# B&R Automation Studio project Task2
Automation Studio 4.9

## Logical view

### Global.typ - Global data types
```iecst
TYPE
	Sys_Handler : 	STRUCT
		Initialize:BOOL:=FALSE;
		Run:BOOL:=FALSE;
		On_Phase_Stop:BOOL:=FALSE;
	END_STRUCT;

	Sub_Sys_Handler : 	STRUCT
		Initialize:BOOL:=FALSE;
		Enable:BOOL:=FALSE;
		Disable:BOOL:=FALSE;
		On_Phase_Stop:BOOL:=FALSE;
	END_STRUCT;

END_TYPE
```

### Global.var - Global variables
```iecst
(* Generic-Axis *)
VAR
	gConveyor : ACP10AXIS_typ;
	gKnife : ACP10AXIS_typ;
END_VAR

(* Logical Buttons*)
VAR
	Init_logical : BOOL;
	Start_logical : BOOL;
	On_Phase_Stop_logical : BOOL;
	Trigger_logical : BOOL;
	Reset_logical : BOOL;
END_VAR
(* Handlers *)
VAR
	Machine_Handler : Sys_Handler;
	Conveyor_Handler : Sub_Sys_Handler;
	Cutter_Handler : Sub_Sys_Handler;
	Signal_Management_Handler : Sys_Handler;
END_VAR

VAR
	CONVEYOR_VELOCITY : REAL := 100;
	CONVEYOR_MAX_VELOCITY : REAL := 100;
	CUTTER_VELOCITY : REAL := 400;
	CUTTER_MAX_VELOCITY : REAL := 400;
END_VAR
```

### Package Logical/Libraries - Global libraries

### Library Logical/Libraries/gAxis_lib (IEC)

#### Types.typ - Exported data types
```iecst
TYPE
	gAxis_StateType :
		(
		NotPowered,
		WaitPower,
		Powered,
		Ready,
		CommandHandler,
		MoveVelocity,
		CheckVelocity,
		MoveAdditive,
		CheckPosition,
		CamInState,
		CheckCamState,
		Stop
		);
END_TYPE
```

#### Constants.var - Exported constants
```iecst
VAR CONSTANT
	AXIS_NULL_COMMAND : WORD := 0;
	AXIS_MOVE_VELOCITY : WORD := 1;
	AXIS_MOVE_ADDITIVE : WORD := 2;
	AXIS_CAM_IN : WORD := 3;
	AXIS_STOP : WORD := 4;
	STANDSTILL : WORD := 5;
	DISCRETE_MOTION : WORD := 6;
	CONTINOUS_MOTION : WORD := 7;
END_VAR
```

#### gAxis_lib.fun - Exported functions and function blocks
```iecst
FUNCTION_BLOCK gAxis (*TODO: Add your comment here*) (*$GROUP=User,$CAT=User,$GROUPICON=User.png,$CATICON=User.png*)
	VAR_INPUT
		Master : UDINT;
		Slave : UDINT;
		AxisOperation : INT;
		AxisCommand : WORD := 777;
		Distance : REAL;
		Position : REAL;
		Velocity : REAL;
		Acceleration : REAL;
		Deceleration : REAL;
		Jerk : REAL;
		Direction : USINT;
		ArraySize : INT;
		Scale : REAL;
		Offset : REAL;
		RatioNumerator : INT;
		RatioDenominator : INT;
		CamTableID : USINT;
		MasterScaling : REAL := 360;
		SlaveScaling : REAL := 360;
		MasterOffset : REAL := 10;
		SlaveOffset : REAL := 0;
		StartMode : USINT := 1; (*mcRELATIVE*)
		AxisEnable_in : BOOL;
		Reset : BOOL;
	END_VAR
	VAR_OUTPUT
		ActualPosition : REAL;
		ActualVelocity : REAL;
		AxisEnable_out : BOOL;
		CommandExecuted : BOOL := FALSE;
		CommandAborted : BOOL;
		AxisStatus : WORD;
		AxisError : BOOL;
		AxisErrorID : WORD;
		AxisNotInizialized : BOOL;
	END_VAR
	VAR
		INIT : INT;
		RUN : INT;
		OldDistance : REAL;
		OldVelocity : REAL;
		OldCamTableID : USINT;
		AxisState : gAxis_StateType := NotPowered;
		gA_Power : MC_Power;
		gA_Home : MC_Home;
		gA_MoveVelocity : MC_MoveVelocity;
		gA_MoveAdditive : MC_MoveAdditive;
		gA_CamIn : MC_CamIn;
		gA_CamOut : MC_CamOut;
		gA_ReadActualPosition : MC_ReadActualPosition;
		gA_ReadActualVelocity : MC_ReadActualVelocity;
		gA_ReadAxisError : MC_ReadAxisError;
		gA_ReadStatus : MC_ReadStatus;
		gA_Stop : MC_Stop;
	END_VAR
END_FUNCTION_BLOCK
```

#### gAxis.st
```iecst
(* TODO: Add your comment here *)
FUNCTION_BLOCK gAxis

	CASE AxisState OF

		NotPowered:
			IF AxisEnable_in THEN
				gA_Power.Enable := TRUE;
				AxisState := WaitPower;
			END_IF;

		WaitPower:
			IF gA_Power.Status THEN
				gA_Home.Execute := TRUE;
				(*gA_CamTableSelect.Execute := TRUE;*)
				AxisState := Powered;
			END_IF

		Powered:
			(*IF gA_Home.Done AND gA_CamTableSelect.Done THEN*)

			IF gA_Home.Done THEN
				gA_Home.Execute := FALSE;
				AxisEnable_out := FALSE;
				AxisState := Ready;
			END_IF;

		Ready:
			IF AxisCommand = AXIS_MOVE_VELOCITY THEN
				CommandExecuted := FALSE;
				gA_MoveVelocity.Velocity := Velocity;
				gA_MoveVelocity.Execute := TRUE;
				AxisState := MoveVelocity;
			END_IF;

			IF AxisCommand = AXIS_MOVE_ADDITIVE THEN
				CommandExecuted := FALSE;
				gA_MoveAdditive.Distance := Distance;
				gA_MoveAdditive.Execute := TRUE;
				AxisState := MoveAdditive;
			END_IF;

			IF AxisCommand = AXIS_CAM_IN THEN
				CommandExecuted := FALSE;
				gA_CamIn.Execute := TRUE;
				AxisState := CamInState;
			END_IF

			IF AxisCommand = AXIS_STOP THEN
				CommandExecuted := FALSE;
				gA_Stop.Execute := TRUE;
				AxisState := Stop;
			END_IF;

		MoveVelocity:
			IF gA_MoveVelocity.InVelocity THEN
				OldVelocity := Velocity;
				gA_MoveVelocity.Execute := FALSE;
				CommandExecuted := TRUE;
				AxisState := CheckVelocity;
			END_IF;

			IF AxisCommand <> AXIS_MOVE_VELOCITY THEN
				gA_MoveVelocity.Execute := FALSE;
				CommandExecuted := FALSE;
				AxisState := Ready;
			END_IF;

		CheckVelocity:
			IF Velocity <> OldVelocity THEN
				OldVelocity := Velocity;
				gA_MoveVelocity.Velocity := Velocity;
				gA_MoveVelocity.Execute := TRUE;
				CommandExecuted := FALSE;
				AxisState := MoveVelocity;
			END_IF;

			IF AxisCommand <> AXIS_MOVE_VELOCITY THEN
				gA_MoveVelocity.Execute := FALSE;
				CommandExecuted := FALSE;
				AxisState := Ready;
			END_IF;

		MoveAdditive:
			IF gA_MoveAdditive.Done THEN
				OldDistance := Distance;
				gA_MoveAdditive.Execute := FALSE;
				CommandExecuted := TRUE;
				AxisState := CheckPosition;
			END_IF;

			IF AxisCommand <> AXIS_MOVE_ADDITIVE THEN
				gA_MoveAdditive.Execute := FALSE;
				CommandExecuted := FALSE;
				AxisState := Ready;
			END_IF;

		CheckPosition:
			IF Distance <> OldDistance THEN
				OldDistance := Distance;
				gA_MoveAdditive.Distance := Distance;
				gA_MoveAdditive.Execute := TRUE;
				CommandExecuted := FALSE;
				AxisState := MoveAdditive;
			END_IF;

			IF AxisCommand <> AXIS_MOVE_ADDITIVE THEN
				gA_MoveAdditive.Execute := FALSE;
				CommandExecuted := FALSE;
				AxisState := Ready;
			END_IF;

		CamInState:
			IF gA_CamIn.EndOfProfile THEN
				OldCamTableID := CamTableID;
				gA_CamIn.Execute := FALSE;
				CommandExecuted := TRUE;
				AxisState := CheckCamState;
			END_IF

			IF AxisCommand <> AXIS_CAM_IN THEN
				gA_CamIn.Execute := FALSE;
				CommandExecuted := FALSE;
				AxisState :=  Ready;
			END_IF

		CheckCamState:
			IF CamTableID <> OldCamTableID THEN
				OldCamTableID := CamTableID;
				gA_CamIn.Execute := TRUE;
				CommandExecuted := FALSE;
				AxisState := CamInState;
			END_IF;

			IF AxisCommand <> AXIS_MOVE_ADDITIVE THEN
				gA_CamIn.Execute := FALSE;
				CommandExecuted := FALSE;
				AxisState := Ready;
			END_IF;

		Stop:
			IF (gA_Stop.Done) THEN
				CommandExecuted := TRUE;
			END_IF

			IF (AxisCommand <> AXIS_STOP ) THEN
				gA_Stop.Execute := FALSE;
				CommandExecuted := FALSE;

				AxisState := Ready;
			END_IF

	END_CASE;

	AxisEnable_in := AxisEnable_out;

	gA_Power.Axis := Slave;
	gA_Power();

	gA_Home.Axis := Slave;
	gA_Home.Position := Position;
	gA_Home();

	(*
	gA_CamTableSelect.Master := Master;
	gA_CamTableSelect.Slave := Slave;
	gA_CamTableSelect.CamTable := 'Cam';
	gA_CamTableSelect.Periodic := mcNON_PERIODIC;
	gA_CamTableSelect();
	CamTableID := gA_CamTableSelect.CamTableID;
	*)

	gA_MoveVelocity.Axis := Slave;
	gA_MoveVelocity.Velocity := Velocity;
	gA_MoveVelocity.Acceleration := Acceleration;
	gA_MoveVelocity.Deceleration := Deceleration;
	gA_MoveVelocity();

	IF OldDistance = 0 THEN
		OldDistance := Distance;
	END_IF;

	gA_MoveAdditive.Axis := Slave;
	gA_MoveAdditive.Distance := Distance;
	gA_MoveAdditive.Velocity := Velocity;
	gA_MoveAdditive.Acceleration := Acceleration;
	gA_MoveAdditive.Deceleration := Deceleration;
	gA_MoveAdditive();

	gA_ReadActualPosition.Axis := Slave;
	gA_ReadActualPosition.Enable := TRUE;
	gA_ReadActualPosition();

	ActualPosition := gA_ReadActualPosition.Position;

	gA_ReadActualVelocity.Axis := Slave;
	gA_ReadActualVelocity.Enable := TRUE;
	gA_ReadActualVelocity();

	ActualVelocity := gA_ReadActualVelocity.Velocity;

	gA_CamIn.CamTableID := CamTableID;
	gA_CamIn.StartMode := StartMode;
	gA_CamIn.MasterScaling := MasterScaling;
	gA_CamIn.SlaveScaling := SlaveScaling;
	gA_CamIn.MasterOffset := MasterOffset;
	gA_CamIn.SlaveOffset := SlaveOffset;
	gA_CamIn(Master := Master, Slave := Slave);

	gA_CamOut(Slave:=Slave);

	gA_Stop.Axis := Slave;
	gA_Stop.Deceleration := Deceleration;
	gA_Stop();

	gA_ReadStatus.Enable := TRUE;
	gA_ReadStatus.Axis := Slave;
	gA_ReadStatus();

	IF gA_ReadStatus.StandStill THEN
		AxisStatus := STANDSTILL;
	END_IF;

	IF gA_ReadStatus.DiscreteMotion THEN
		AxisStatus := DISCRETE_MOTION;
	END_IF;

	IF gA_ReadStatus.ContinuousMotion THEN
		AxisStatus := CONTINOUS_MOTION;
	END_IF;

END_FUNCTION_BLOCK
```

### Library Logical/Libraries/filter_lib (IEC)

#### filter.st
```iecst
(* TODO: Add your comment here *)
FUNCTION_BLOCK filter

	IF Delay > 0 THEN
		Delay := Delay -1;
	END_IF;

	IF Delay = 0 THEN
	  DelayedSignal := Signal;
	END_IF;

	IF Signal = DelayedSignal THEN

		IF Signal THEN
			Delay := DeactivationDelay;
		ELSE
			Delay := ActivationDelay;
		END_IF;

	END_IF;
END_FUNCTION_BLOCK
```

- Visualisation Logical/mappView (not shown)


- Data object Logical/gConveyorobj/gConveyora (Apt) (no source held here)

### Package Logical/gKnifeobj - gKnifeobj

- Data object Logical/gKnifeobj/gKnifea (Apt) (no source held here)

### Data object Logical/gKnifeobj/gKnifei (Ax)

#### gKnifei.ax
```
InitParameter (Version=5.16.2, NcSwId=Acp10)
  ACP10AXIS_typ:
    dig_in:
      level:
        reference = ncACTIV_HI
        pos_hw_end = ncACTIV_HI
        neg_hw_end = ncACTIV_HI
        trigger1 = ncACTIV_HI
        trigger2 = ncACTIV_HI
    encoder_if:
      parameter:
        count_dir = ncSTANDARD
        scaling:
          load:
            units = 360
            rev_motor = 1
    limit:
      parameter:
        v_pos = 10000
        v_neg = 10000
        a1_pos = 50000
        a2_pos = 50000
        a1_neg = 50000
        a2_neg = 50000
        t_jolt = 0
        t_in_pos = 0
        pos_sw_end = 2000000000
        neg_sw_end = -2000000000
        ds_warning = 500
        ds_stop = 1000
        a_stop = 1.0e30
        dv_stop = 0
        dv_stop_mode = ncOFF
    controller:
      mode = ncPOSITION
      position:
        kv = 50
        tn = 0
        t_predict = 0.0004
        t_total = 0.0004
        p_max = 1.0e30
        i_max = 0
      speed:
        kv = 2.0
        tn = 0
        t_filter = 0.0
        isq_filter1:
          type = ncOFF
          a0 = 0.0
          a1 = 0.0
          b0 = 0.0
          b1 = 0.0
          b2 = 0.0
          c0_par_id = 0
          c1_par_id = 0
        isq_filter2:
          type = ncOFF
          a0 = 0.0
          a1 = 0.0
          b0 = 0.0
          b1 = 0.0
          b2 = 0.0
          c0_par_id = 0
          c1_par_id = 0
        isq_filter3:
          type = ncOFF
          a0 = 0.0
          a1 = 0.0
          b0 = 0.0
          b1 = 0.0
          b2 = 0.0
          c0_par_id = 0
          c1_par_id = 0
      uf:
        type = ncLINEAR + ncCORRECTION
        auto_config = ncMOTOR_PAR
        u0 = 0
        un = 0
        fn = 50.0
        k_f_slip = 0
      ff:
        mode = ncSTANDARD
        torque_load = 0.0
        torque_pos = 0.0
        torque_neg = 0.0
        kv_torque = 0.0
        inertia = 0.0
        t_filter_a = 0.0
      fb:
        mode = ncSTANDARD
        speed_mix_ratio = 0.0
        speed_kv = 2.0
      model:
        mass1:
          inertia = 0
          viscous_friction = 0
        mass2:
          inertia = 0
          viscous_friction = 0
          stiffness = 0
          damping = 0
    move:
      stop:
        parameter[0]:
          decel_ramp = ncA_LIMIT
          controller = ncON
        parameter[1]:
          decel_ramp = ncA_LIMIT
          controller = ncON
        parameter[2]:
          decel_ramp = ncA_LIMIT
          controller = ncON
        parameter[3]:
          decel_ramp = ncA_LIMIT
          controller = ncON
        quickstop:
          decel_ramp = ncA_LIMIT
          t_jolt = 0
        drive_error:
          decel_ramp = ncA_LIMIT
      homing:
        parameter:
          s = 0
          v_switch = 5000
          v_trigger = 500
          a = 50000
          mode = ncDIRECT
          edge_sw = ncPOSITIVE
          start_dir = ncPOSITIVE
          trigg_dir = ncPOSITIVE
          ref_pulse = ncOFF
          fix_dir = ncOFF
          tr_s_block = 0
          torque_lim = 0
          ds_block = 0
          ds_stop = 0
      basis:
        parameter:
          v_pos = 5000
          v_neg = 5000
          a1_pos = 50000
          a2_pos = 50000
          a1_neg = 50000
          a2_neg = 50000
    message:
      text:
        parameter:
          format = ncBREAK
          columns = 80
          data_modul = acp10etxen
```

### Data object Logical/Cam (Cam)

#### Cam.cam
```
CamProfile (NcSwId=ACP10, MasterAxisVelocity=1, MasterAxisAcceleration=0, DefaultCurveType=Polynomial5, MathematicalNotation=true)
  FixPoint (x=0, IsMathX=true, y=0, IsDefinedDy=false, Dy=0, IsMathDy=true, IsDefinedDdy=false, Ddy=0, IsMathDdy=true, IsDefinedDddy=false, Dddy=0, IsMathDddy=true)
  FixPoint (x=0.5, IsMathX=true, y=0, IsDefinedDy=false, Dy=0, IsMathDy=true, IsDefinedDdy=false, Ddy=0, IsMathDdy=true, IsDefinedDddy=false, Dddy=0, IsMathDddy=true)
  FixPoint (x=0.55, IsMathX=true, y=0.5, IsDefinedDy=false, Dy=0, IsMathDy=true, IsDefinedDdy=false, Ddy=0, IsMathDdy=true, IsDefinedDddy=false, Dddy=0, IsMathDddy=true)
  FixPoint (x=0.6, IsMathX=true, y=0, IsDefinedDy=false, Dy=0, IsMathDy=true, IsDefinedDdy=false, Ddy=0, IsMathDdy=true, IsDefinedDddy=false, Dddy=0, IsMathDddy=true)
  FixPoint (x=1, IsMathX=true, y=0, IsDefinedDy=false, Dy=0, IsMathDy=true, IsDefinedDdy=false, Ddy=0, IsMathDdy=true, IsDefinedDddy=false, Dddy=0, IsMathDddy=true)
  Curve (Type=Polynomial5)
    LeftBoundary (IsDefinedDdy=false, Ddy=0, IsMathDdy=true, IsDefinedDddy=false, Dddy=0, IsMathDddy=true)
    RightBoundary (IsDefinedDdy=false, Ddy=0, IsMathDdy=true, IsDefinedDddy=false, Dddy=0, IsMathDddy=true)
    Spline3 (IsContinuous4Derivative=false, IsDefinedSaddlePoint=false, IsDefinedLineAs2ndSegment=false, IsDefinedSlopeOfLine=false, SlopeOfLine=0, IsMathSlopeOfLine=true)
    Supremum (y=1.7e+308, Dy=1.7e+308, IsMathDy=true, Ddy=1.7e+308, IsMathDdy=true, Dddy=1.7e+308, IsMathDddy=true)
    Infimum (y=-1.7e+308, Dy=-1.7e+308, IsMathDy=true, Ddy=-1.7e+308, IsMathDdy=true, Dddy=-1.7e+308, IsMathDddy=true)
  Curve (Type=Polynomial5)
    LeftBoundary (IsDefinedDdy=false, Ddy=0, IsMathDdy=true, IsDefinedDddy=false, Dddy=0, IsMathDddy=true)
    RightBoundary (IsDefinedDdy=false, Ddy=0, IsMathDdy=true, IsDefinedDddy=false, Dddy=0, IsMathDddy=true)
    Spline3 (IsContinuous4Derivative=false, IsDefinedSaddlePoint=false, IsDefinedLineAs2ndSegment=false, IsDefinedSlopeOfLine=false, SlopeOfLine=0, IsMathSlopeOfLine=true)
    Supremum (y=1.7e+308, Dy=1.7e+308, IsMathDy=true, Ddy=1.7e+308, IsMathDdy=true, Dddy=1.7e+308, IsMathDddy=true)
    Infimum (y=-1.7e+308, Dy=-1.7e+308, IsMathDy=true, Ddy=-1.7e+308, IsMathDdy=true, Dddy=-1.7e+308, IsMathDddy=true)
  Curve (Type=Polynomial5)
    LeftBoundary (IsDefinedDdy=false, Ddy=0, IsMathDdy=true, IsDefinedDddy=false, Dddy=0, IsMathDddy=true)
    RightBoundary (IsDefinedDdy=false, Ddy=0, IsMathDdy=true, IsDefinedDddy=false, Dddy=0, IsMathDddy=true)
    Spline3 (IsContinuous4Derivative=false, IsDefinedSaddlePoint=false, IsDefinedLineAs2ndSegment=false, IsDefinedSlopeOfLine=false, SlopeOfLine=0, IsMathSlopeOfLine=true)
    Supremum (y=1.7e+308, Dy=1.7e+308, IsMathDy=true, Ddy=1.7e+308, IsMathDdy=true, Dddy=1.7e+308, IsMathDddy=true)
    Infimum (y=-1.7e+308, Dy=-1.7e+308, IsMathDy=true, Ddy=-1.7e+308, IsMathDdy=true, Dddy=-1.7e+308, IsMathDddy=true)
  Curve (Type=Polynomial5)
    LeftBoundary (IsDefinedDdy=false, Ddy=0, IsMathDdy=true, IsDefinedDddy=false, Dddy=0, IsMathDddy=true)
    RightBoundary (IsDefinedDdy=false, Ddy=0, IsMathDdy=true, IsDefinedDddy=false, Dddy=0, IsMathDddy=true)
    Spline3 (IsContinuous4Derivative=false, IsDefinedSaddlePoint=false, IsDefinedLineAs2ndSegment=false, IsDefinedSlopeOfLine=false, SlopeOfLine=0, IsMathSlopeOfLine=true)
    Supremum (y=1.7e+308, Dy=1.7e+308, IsMathDy=true, Ddy=1.7e+308, IsMathDdy=true, Dddy=1.7e+308, IsMathDddy=true)
    Infimum (y=-1.7e+308, Dy=-1.7e+308, IsMathDy=true, Ddy=-1.7e+308, IsMathDdy=true, Dddy=-1.7e+308, IsMathDddy=true)
  Cam (LeftBoundaryIndex=0, RightBoundaryIndex=4)
    Supremum (y=1.7e+308, Dy=1.7e+308, IsMathDy=true, Ddy=1.7e+308, IsMathDdy=true, Dddy=1.7e+308, IsMathDddy=true)
    Infimum (y=-1.7e+308, Dy=-1.7e+308, IsMathDy=true, Ddy=-1.7e+308, IsMathDdy=true, Dddy=1.7e+308, IsMathDddy=true)
  ChartExtensions
```

### Program Logical/Main (IEC)

#### Types.typ
```iecst
TYPE
	Main_States: (
		Main_ready_to_be_initialized,
		Main_initializing,
		Main_ready_to_run,
		Main_running,
		Main_on_phase_stopping
	);
END_TYPE
```

#### Main.st
```iecst
PROGRAM _CYCLIC
	(* Insert code here *)

	CASE state OF
		Main_ready_to_be_initialized:
			IF Init_logical THEN
				Machine_Handler.Initialize := TRUE;

				state := Main_initializing;
			END_IF;

		Main_initializing:
			IF NOT Machine_Handler.Initialize THEN

				state := Main_ready_to_run;
			END_IF;

		Main_ready_to_run:
			IF Start_logical THEN
				Machine_Handler.Run := TRUE;

				state := Main_running;
			END_IF;

		Main_running:
			IF On_Phase_Stop_logical THEN
				Machine_Handler.Run := FALSE;
				Machine_Handler.On_Phase_Stop := TRUE;

				state := Main_on_phase_stopping;
			END_IF;

		Main_on_phase_stopping:
			IF NOT On_Phase_Stop_logical THEN
				Machine_Handler.On_Phase_Stop := FALSE;

				state := Main_ready_to_run;
			END_IF;
	END_CASE;

END_PROGRAM
```

### Program Logical/MachineProgram (IEC)

#### Types.typ
```iecst
TYPE
	Machine_States: (
					Machine_ready_to_be_initialized,
					Machine_initializing,
					Machine_ready_to_run,
					Conveyor_Enabling,
					Cutter_Enabling,
					Machine_on_phase_stopping);
END_TYPE
```

#### Variables.var
```iecst
VAR
	state: Machine_States := Machine_ready_to_be_initialized;
END_VAR
```

#### Main.st
```iecst
PROGRAM _CYCLIC
	(* Insert code here *)
	CASE state OF

		Machine_ready_to_be_initialized:
			IF Machine_Handler.Initialize THEN
				Conveyor_Handler.Initialize := TRUE;
				Cutter_Handler.Initialize := TRUE;

				state := Machine_initializing;
			END_IF;

		Machine_initializing:
			IF NOT Conveyor_Handler.Initialize AND NOT Cutter_Handler.Initialize THEN
				Machine_Handler.Initialize := FALSE;

				state := Machine_ready_to_run;
			END_IF;

		Machine_ready_to_run:
			IF Machine_Handler.Run THEN
				Conveyor_Handler.Enable := TRUE;

				state := Conveyor_Enabling;
			END_IF;

		Conveyor_Enabling:
			IF Machine_Handler.On_Phase_Stop THEN
				Conveyor_Handler.On_Phase_Stop := TRUE;
				Cutter_Handler.On_Phase_Stop := TRUE;

				state := Machine_on_phase_stopping;

			ELSIF NOT Conveyor_Handler.Enable AND Trigger_logical THEN
				Cutter_Handler.Enable := TRUE;

				state := Cutter_Enabling;
			END_IF;

		Cutter_Enabling:
			IF NOT Cutter_Handler.Enable THEN

				state := Conveyor_Enabling;
			END_IF;

		Machine_on_phase_stopping:
			IF NOT Machine_Handler.On_Phase_Stop THEN
				Conveyor_Handler.On_Phase_Stop := FALSE;
				Cutter_Handler.On_Phase_Stop := FALSE;

				state := Machine_ready_to_run;
			END_IF;
	END_CASE;

END_PROGRAM

PROGRAM _EXIT
	(* Insert code here *)

END_PROGRAM
```

### Program Logical/Conveyor (IEC)

#### Types.typ
```iecst
TYPE
	Conveyor_States: (
		Conveyor_ready_to_be_initialized,
		Conveyor_initializing,
		Conveyor_ready_to_be_enabled,
		Conveyor_enabling,
		Conveyor_ready_to_be_disabled,
		Conveyor_on_phase_stopping
	);
END_TYPE
```

#### Variables.var
```iecst
VAR
	Conveyor : gAxis;
END_VAR

VAR
	state: Conveyor_States := Conveyor_ready_to_be_initialized;
END_VAR

VAR
	Axis_Command : WORD := AXIS_NULL_COMMAND;
	Axis_Command_Executed : BOOL;
	Axis_Enable : BOOL;
END_VAR

VAR
	CONVEYOR_POSITION : REAL;
	CONVEYOR_ACTUAL_VELOCITY : INT;
	CONVEYOR_ACCELLERATION : REAL := 100;
	CONVEYOR_DEACCELLERATION : REAL := 100;
	CONVEYOR_DISTANCE : REAL := 100;
END_VAR

VAR CONSTANT
	AXIS_NULL_COMMAND : WORD := 0;
	AXIS_MOVE_VELOCITY : WORD := 1;
	AXIS_MOVE_ADDITIVE : WORD := 2;
	AXIS_CAM_IN : WORD := 3;
	AXIS_STOP : WORD := 4;
END_VAR
```

#### Main.st
```iecst
PROGRAM _INIT
	(* Insert code here *)

END_PROGRAM

PROGRAM _CYCLIC
	(* Insert code here *)
	CASE state OF
		Conveyor_ready_to_be_initialized:
			IF Conveyor_Handler.Initialize THEN
				Axis_Enable := TRUE;

				state := Conveyor_initializing;
			END_IF;

		Conveyor_initializing:
			IF NOT Axis_Enable THEN
				Conveyor_Handler.Initialize := FALSE;

				state := Conveyor_ready_to_be_enabled;
			END_IF;

		Conveyor_ready_to_be_enabled:
			IF Conveyor_Handler.Enable THEN
				Axis_Command := AXIS_MOVE_VELOCITY;

				state := Conveyor_enabling;
			END_IF;

		Conveyor_enabling:
			IF Axis_Command_Executed THEN
				Conveyor_Handler.Enable := FALSE;

				state := Conveyor_ready_to_be_disabled;
			END_IF;

		Conveyor_ready_to_be_disabled:
			IF Conveyor_Handler.On_Phase_Stop THEN
				Axis_Command := AXIS_STOP;

				state := Conveyor_on_phase_stopping;
			END_IF;

		Conveyor_on_phase_stopping:
			IF NOT Conveyor_Handler.On_Phase_Stop THEN

				state := Conveyor_ready_to_be_enabled;
			END_IF;
	END_CASE;

	Conveyor.Slave	:= ADR(gConveyor);

	Conveyor.AxisEnable_in := Axis_Enable;
	Conveyor.AxisCommand := Axis_Command;

	Conveyor.Velocity	:= CONVEYOR_VELOCITY;
	Conveyor.Acceleration	:= CONVEYOR_ACCELLERATION;
	Conveyor.Deceleration	:= CONVEYOR_DEACCELLERATION;

	Conveyor();

	Axis_Enable := Conveyor.AxisEnable_out;
	Axis_Command_Executed := Conveyor.CommandExecuted;
	CONVEYOR_POSITION := Conveyor.ActualPosition;
	CONVEYOR_ACTUAL_VELOCITY := REAL_TO_INT(Conveyor.ActualVelocity);

	ComTCP_SimOutputs.Shaft_0_ACT_POS := CONVEYOR_POSITION;

END_PROGRAM

PROGRAM _EXIT
	(* Insert code here *)

END_PROGRAM
```

### Program Logical/Knife (IEC)

#### Types.typ
```iecst
TYPE
	Cutter_States:
		(
		Cutter_ready_to_be_initialized,
		Cutter_initializing,
		Cutter_ready_to_be_enabled,
		Cutter_enabling
	);
END_TYPE
```

#### Variables.var
```iecst
VAR
	Knife : gAxis;
	CamTableSelect : MC_CamTableSelect;
	CamTableID : USINT;

END_VAR

VAR
	state: Cutter_States := Cutter_ready_to_be_initialized;
END_VAR

VAR
	Axis_Command : WORD := AXIS_NULL_COMMAND;
	Axis_Command_Executed : BOOL;
	Axis_Enable : BOOL;
END_VAR

VAR
	CUTTER_POSITION : REAL;
	CUTTER_ACTUAL_VELOCITY : REAL;
	CUTTER_ACCELLERATION : REAL := 400;
	CUTTER_DEACCELLERATION : REAL := 400;
END_VAR

VAR CONSTANT
	AXIS_NULL_COMMAND : WORD := 0;
	AXIS_MOVE_VELOCITY : WORD := 1;
	AXIS_MOVE_ADDITIVE : WORD := 2;
	AXIS_CAM_IN : WORD := 3;
	AXIS_STOP : WORD := 4;
END_VAR
```

#### Main.st
```iecst
PROGRAM _INIT
	(* Insert code here *)

END_PROGRAM

PROGRAM _CYCLIC
	(* Insert code here *)

	CASE state OF

		Cutter_ready_to_be_initialized:
			IF Cutter_Handler.Initialize THEN
				Axis_Enable := TRUE;
				CamTableSelect.Execute := TRUE;

				state := Cutter_initializing;
			END_IF;

		Cutter_initializing:
			IF NOT Axis_Enable AND CamTableSelect.Done THEN
				Cutter_Handler.Initialize := FALSE;
				CamTableID := CamTableSelect.CamTableID;
				CamTableSelect.Execute := FALSE;

				state := Cutter_ready_to_be_enabled;
			END_IF;

		Cutter_ready_to_be_enabled:
			IF Cutter_Handler.Enable THEN
				Axis_Command := AXIS_CAM_IN;

				state := Cutter_enabling;
			END_IF;

		Cutter_enabling:
			IF Axis_Command_Executed THEN
				Axis_Command := AXIS_NULL_COMMAND;
				Cutter_Handler.Enable := FALSE;

				state := Cutter_ready_to_be_enabled;
			END_IF;

	END_CASE;

	CamTableSelect.Master := ADR(gConveyor);
	CamTableSelect.Slave := ADR(gKnife);
	CamTableSelect.CamTable := 'Cam';
	CamTableSelect.Periodic := mcNON_PERIODIC;
	CamTableSelect();

	Knife.Master	:= ADR(gConveyor);
	Knife.Slave	:= ADR(gKnife);

	Knife.AxisEnable_in := Axis_Enable;
	Knife.AxisCommand := Axis_Command;

	Knife.CamTableID := CamTableID;
	Knife.Velocity := CUTTER_VELOCITY;
	Knife.Acceleration	:= CUTTER_ACCELLERATION;
	Knife.Deceleration	:= CUTTER_DEACCELLERATION;

	Knife();

	Axis_Enable := Knife.AxisEnable_out;
	Axis_Command_Executed := Knife.CommandExecuted;
	CUTTER_POSITION	:= Knife.ActualPosition;
	CUTTER_ACTUAL_VELOCITY:= Knife.ActualVelocity;

	ComTCP_SimOutputs.Shaft_1_ACT_POS := CUTTER_POSITION;

END_PROGRAM

PROGRAM _EXIT
	(* Insert code here *)

END_PROGRAM
```

### Program Logical/ISP (IEC)

#### Variables.var
```iecst
(* Phisical Buttons*)
VAR
	DI1 : BOOL;
	DI2 : BOOL;
	DI3 : BOOL;
	DI4 : BOOL;
	DI5 : BOOL;
	DI6 : BOOL;
	P1 : INT;
	P2 : INT;
END_VAR

(* HMI PANEL *)
VAR
	INIT_HMI : BOOL;
	START_HMI : BOOL;
	STOP_HMI : BOOL;
	TRIGGER_HMI : BOOL;
	RESET_HMI : BOOL;
	SIM_ON_HMI : BOOL;
	CONVEYOR_SPEED_HMI : UINT;
	CUTTER_SPEED_HMI : UINT;
END_VAR

(* Filters *)
VAR
	DI1_filter : filter;
	DI2_filter : filter;
	DI3_filter : filter;
	DI4_filter : filter;
	DI5_filter : filter;
	DI6_filter : filter;
END_VAR

(* DELAY *)
VAR CONSTANT
	DI1_delay : UDINT := 2;
	DI2_delay : UDINT := 2;
	DI3_delay : UDINT := 2;
	DI4_delay : UDINT := 2;
	DI5_delay : UDINT := 2;
	DI6_delay : UDINT := 2;
END_VAR
```

#### Main.st
```iecst
PROGRAM _INIT
	(* Insert code here *)

END_PROGRAM

PROGRAM _CYCLIC
	(* Insert code here *)

	DI1_filter.Signal := DI1;
	DI1_filter.ActivationDelay := DI1_delay;
	DI1_filter.DeactivationDelay := DI1_delay;
	DI1_filter();

	DI3_filter.Signal := DI3;
	DI3_filter.ActivationDelay := DI3_delay;
	DI3_filter.DeactivationDelay := DI3_delay;
	DI3_filter();

	DI4_filter.Signal := DI4;
	DI4_filter.ActivationDelay := DI4_delay;
	DI4_filter.DeactivationDelay := DI4_delay;
	DI4_filter();

	DI5_filter.Signal := DI5;
	DI5_filter.ActivationDelay := DI5_delay;
	DI5_filter.DeactivationDelay := DI5_delay;
	DI5_filter();

	DI6_filter.Signal := DI6;
	DI6_filter.ActivationDelay := DI6_delay;
	DI6_filter.DeactivationDelay := DI6_delay;
	DI6_filter();

	IF SIM_ON_HMI THEN

		Init_logical := DI1_filter.DelayedSignal OR INIT_HMI;
		Start_logical := DI3_filter.DelayedSignal OR START_HMI;
		On_Phase_Stop_logical := DI4_filter.DelayedSignal OR STOP_HMI;
		Trigger_logical := DI5_filter.DelayedSignal OR TRIGGER_HMI;
		Reset_logical := DI6_filter.DelayedSignal OR RESET_HMI;

		CONVEYOR_VELOCITY := UINT_TO_REAL(CONVEYOR_SPEED_HMI)*CONVEYOR_MAX_VELOCITY/(65535);
		CUTTER_VELOCITY := UINT_TO_REAL(CUTTER_SPEED_HMI)*CUTTER_MAX_VELOCITY/(65535);
	ELSE
		Init_logical := DI1_filter.DelayedSignal;
		Start_logical := DI3_filter.DelayedSignal;
		On_Phase_Stop_logical := DI4_filter.DelayedSignal;
		Trigger_logical := DI5_filter.DelayedSignal;
		Reset_logical := DI6_filter.DelayedSignal;

		CONVEYOR_VELOCITY := CONVEYOR_MAX_VELOCITY/(32767)*P1;
		CUTTER_VELOCITY := CUTTER_MAX_VELOCITY/(32767)*P2;
	END_IF

END_PROGRAM

PROGRAM _EXIT
	(* Insert code here *)

END_PROGRAM
```

Listed in the project but not available here: Logical/Libraries/filter_lib/Types.typ, Logical/Libraries/filter_lib/Constants.var, Logical/Libraries/filter_lib/filter_lib.fun, Logical/Libraries/filter_lib/BlinkFB.st, Logical/gConveyorobj/gConveyori, Logical/OSP
